PROGRAM MAIN
VAR
END_VAR

END_PROGRAM

(* stored: Version 1.1.0.1
   POU MAIN: Id {a7d96428-2ed9-4645-a534-7d2e3191ad64} *)
